# EPICS autosave request: iocBoot/gmca_23i_ioc2/dbSave/VF_Be_.req
%
% BURT Request File
%
% $(P)VF:Be:  VFM Bender
%

file assy.req ASSY=$(P)VF:Be
file mtr1.req MTR1=$(P)VF:mbe
file drv1.req DRV1=$(P)VF:BE
